FUNCTION F_RoundREAL : REAL
VAR_INPUT
	rValue:					REAL;
	uiDezimalPlace:	UINT;
END_VAR
VAR
	rResult:				REAL;
	uiMultiplier:		UINT := 1;
	i:							UINT;
END_VAR

FOR i := 1 TO uiDezimalPlace BY 1 DO
	uiMultiplier := uiMultiplier * 10;
END_FOR

rResult := TO_REAL(TO_DINT(rValue * uiMultiplier)) / uiMultiplier;

F_RoundREAL := rResult;

END_FUNCTION

(* stored: Version 1.1.0.1, ProductVersion 3.1.4024.12
   POU F_RoundREAL: Id {db918c49-291a-498e-b3e3-c07540be8418}, SpecialFunc None *)
